// TIA Portal V16 export
// export: Created 2021-11-12T13:31:09.0578565Z, ExportSetting WithDefaults, DisplayName Totally Integrated Automation Portal, DisplayVersion V16 Update 3, DisplayName TIA Portal Version Control Interface, DisplayVersion V16 Update 2, DisplayName TIA Portal Openness, DisplayVersion V16 Update 3, DisplayName SINAMICS Startdrive Advanced, DisplayVersion V16 Update 5, DisplayName SINAMICS Startdrive G130, G150, S120, S150, SINAMICS MV, S210, DisplayVersion V16 Update 5, DisplayName SINAMICS Startdrive G110M, G120, G120C, G120D, G120P, G115D, DisplayVersion V16 Update 5, DisplayName STEP 7 Professional, DisplayVersion V16 Update 3, DisplayName STEP 7 Safety, DisplayVersion V16, DisplayName WinCC UA Professional, DisplayVersion V16 Update 3
FUNCTION_BLOCK "Sfty_Input"   // FB67, F_LAD
{ S7_Optimized_Access := 'TRUE' }
VERSION : 0.1
// Digital and profisafe inputs reading
// stored: AutoNumber true, IsIECCheckEnabled false, UDAEnableTagReadback false
   VAR
      SF_KAS1 { S7_SetPoint := 'True'} : ESTOP1;   // Emergency stop - saw KAS1
      SF_KAS2 { S7_SetPoint := 'True'} : ESTOP1;   // Emergency stop - saw KAS2
      SF_BSN1_2 { S7_SetPoint := 'True'} : ESTOP1;   // Emergency stop - owen BSN1 / BSN2
      SF_SCH1 { S7_SetPoint := 'True'} : ESTOP1;   // Emergency stop - press SCH1
      SF_BSN3 { S7_SetPoint := 'True'} : ESTOP1;   // Emergency stop - owen BSN3
      SF_BSN4_5 { S7_SetPoint := 'True'} : ESTOP1;   // Emergency stop - owen BSN4 / BSN5
      SF_THM1 { S7_SetPoint := 'True'} : ESTOP1;   // Emergency stop - blaster THM1
      SF_THM2 { S7_SetPoint := 'True'} : ESTOP1;   // Emergency stop - blaster THM2
      "SF_1R1-RC01" { S7_SetPoint := 'True'} : ESTOP1;   // Emergency stop - robot 1R1-RC01
      "SF_1R2-RC01" { S7_SetPoint := 'True'} : ESTOP1;   // Emergency stop - robot 1R2-RC01
      "SF_1R3-RC01" { S7_SetPoint := 'True'} : ESTOP1;   // Emergency stop - robot 1R3-RC01
      "SF_1R4-RC01" { S7_SetPoint := 'True'} : ESTOP1;   // Emergency stop - robot 1R4-RC01
      "SF_1R5-RC01" { S7_SetPoint := 'True'} : ESTOP1;   // Emergency stop - robot 1R5-RC01
      "SF_1R6-RC01" { S7_SetPoint := 'True'} : ESTOP1;   // Emergency stop - robot 1R6-RC01
      "SF_2R1-RC01" { S7_SetPoint := 'True'} : ESTOP1;   // Emergency stop - robot 2R1-RC01
      "SF_2R2-RC01" { S7_SetPoint := 'True'} : ESTOP1;   // Emergency stop - robot 2R2-RC01
      "SF_000UH11-SF01_12" { S7_SetPoint := 'True'} : ESTOP1;   // Emergency stop button - panel 000+UH11
      "SF_000UH10-SF01_12" { S7_SetPoint := 'True'} : ESTOP1;   // Emergency stop button - panel 000+UH10
      "SF_100UH11-SF01_12" { S7_SetPoint := 'True'} : ESTOP1;   // Emergency stop button - panel 100+UH11
      "SF_100UH12-SF01_12" { S7_SetPoint := 'True'} : ESTOP1;   // Emergency stop button - panel 100+UH12
      "SF_100UH13-SF01_12" { S7_SetPoint := 'True'} : ESTOP1;   // Emergency stop button - panel 100+UH13
      "SF_100UF01-SF01_12" { S7_SetPoint := 'True'} : ESTOP1;   // Emergency stop button - panel 100+UF01
      "SF_200UH11-SF01_12" { S7_SetPoint := 'True'} : ESTOP1;   // Emergency stop button - panel 200+UH11
      "SF_200UF01-SF01_12" { S7_SetPoint := 'True'} : ESTOP1;   // Emergency stop button - panel 200+UF01
      "SF_210UF01-SF01_12" { S7_SetPoint := 'True'} : ESTOP1;   // Emergency stop button - panel 210+UF01
      "SF_220UF01-SF01_12" { S7_SetPoint := 'True'} : ESTOP1;   // Emergency stop button - panel 220+UF01
      "SF_230UF01-SF01_12" { S7_SetPoint := 'True'} : ESTOP1;   // Emergency stop button - panel 230+UF01
      "SF_300UH11-SF01_12" { S7_SetPoint := 'True'} : ESTOP1;   // Emergency stop button - panel 300+UH11
      "SF_310UH31-SF01_12" { S7_SetPoint := 'True'} : ESTOP1;   // Emergency stop button - panel 300+UH11
      "SF_330UF01-SF01_12" { S7_SetPoint := 'True'} : ESTOP1;   // Emergency stop button - panel 330+UF01
      "SF_400UH11-SF01_12" { S7_SetPoint := 'True'} : ESTOP1;   // Emergency stop button - panel 400+UH11
      "SF_400UH31-SF01_12" { S7_SetPoint := 'True'} : ESTOP1;   // Emergency stop button - panel 400+UH31
      "SF_410UH31-SF01_12" { S7_SetPoint := 'True'} : ESTOP1;   // Emergency stop button - panel 400+UH31
      "SF_420UH31-SF01_12" { S7_SetPoint := 'True'} : ESTOP1;   // Emergency stop button - panel 400+UH31
      "SF_100+RU01-QQ01" { S7_SetPoint := 'True'} : ESTOP1;   // Emergency stop button - gate 100+RU01-QQ01
      "SF_100+RU01-QQ02" { S7_SetPoint := 'True'} : ESTOP1;   // Emergency stop button - gate 100+RU01-QQ02
      "SF_100+RU01-QQ03" { S7_SetPoint := 'True'} : ESTOP1;   // Emergency stop button - gate 100+RU01-QQ03
      "SF_100+RU01-QQ04" { S7_SetPoint := 'True'} : ESTOP1;   // Emergency stop button - gate 100+RU01-QQ04
      "SF_100+RU01-QQ05" { S7_SetPoint := 'True'} : ESTOP1;   // Emergency stop button - gate 100+RU01-QQ05
      "SF_100+RU01-QQ06" { S7_SetPoint := 'True'} : ESTOP1;   // Emergency stop button - gate 100+RU01-QQ06
      "SF_100+RU01-QQ07" { S7_SetPoint := 'True'} : ESTOP1;   // Emergency stop button - gate 100+RU01-QQ07
      "SF_100+RU01-QQ08" { S7_SetPoint := 'True'} : ESTOP1;   // Emergency stop button - gate 100+RU01-QQ08
      "SF_200RU01-QQ01" { S7_SetPoint := 'True'} : ESTOP1;   // Emergency stop button - gate 200RU01-QQ01
      "SF_200RU01-QQ02" { S7_SetPoint := 'True'} : ESTOP1;   // Emergency stop button - gate 200RU01-QQ02
      "SF_200RU01-QQ03" { S7_SetPoint := 'True'} : ESTOP1;   // Emergency stop button - gate 200RU01-QQ03
      "SF_200RU01-QQ04" { S7_SetPoint := 'True'} : ESTOP1;   // Emergency stop button - gate 200RU01-QQ04
      "SF_200RU01-QQ05" { S7_SetPoint := 'True'} : ESTOP1;   // Emergency stop button - gate 200RU01-QQ05
      "SF_100+RU01-QQ01_lock" { S7_SetPoint := 'True'} : ESTOP1;   // Gate is closed and locked - 100+RU01-QQ01
      "SF_100+RU01-QQ02_lock" { S7_SetPoint := 'True'} : ESTOP1;   // Gate is closed and locked - 100+RU01-QQ02
      "SF_100+RU01-QQ03_lock" { S7_SetPoint := 'True'} : ESTOP1;   // Gate is closed and locked - 100+RU01-QQ03
      "SF_100+RU01-QQ04_lock" { S7_SetPoint := 'True'} : ESTOP1;   // Gate is closed and locked - 100+RU01-QQ04
      "SF_100+RU01-QQ05_lock" { S7_SetPoint := 'True'} : ESTOP1;   // Gate is closed and locked - 100+RU01-QQ05
      "SF_100+RU01-QQ06_lock" { S7_SetPoint := 'True'} : ESTOP1;   // Gate is closed and locked - 100+RU01-QQ06
      "SF_100+RU01-QQ07_lock" { S7_SetPoint := 'True'} : ESTOP1;   // Gate is closed and locked - 100+RU01-QQ07
      "SF_100+RU01-QQ08_lock" { S7_SetPoint := 'True'} : ESTOP1;   // Gate is closed and locked - 100+RU01-QQ08
      "SF_200RU01-QQ01_lock" { S7_SetPoint := 'True'} : ESTOP1;   // Gate is closed and locked - 200RU01-QQ01
      "SF_200RU01-QQ02_lock" { S7_SetPoint := 'True'} : ESTOP1;   // Gate is closed and locked - 200RU01-QQ02
      "SF_200RU01-QQ03_lock" { S7_SetPoint := 'True'} : ESTOP1;   // Gate is closed and locked - 200RU01-QQ03
      "SF_200RU01-QQ04_lock" { S7_SetPoint := 'True'} : ESTOP1;   // Gate is closed and locked - 200RU01-QQ04
      "SF_200RU01-QQ05_lock" { S7_SetPoint := 'True'} : ESTOP1;   // Gate is closed and locked - 200RU01-QQ05
      "SF_100+RU01-BG01_close" { S7_SetPoint := 'True'} : ESTOP1;   // Fence closed - 100+RU01-BG01
      "SF_100+RU01-BG02_close" { S7_SetPoint := 'True'} : ESTOP1;   // Fence closed - 100+RU01-BG02
      "SF_200RU01-BG01_close" { S7_SetPoint := 'True'} : ESTOP1;   // Fence closed - 200RU01-BG01
      "SF_100UR01-KG01R" { S7_SetPoint := 'True'} : ESTOP1;   // Light barrier ok - 100UR01-KG01
      "SF_100UR01-KG02R" { S7_SetPoint := 'True'} : ESTOP1;   // Light barrier ok - 100UR01-KG02
   END_VAR
BEGIN

REGION Network 1: *************** Estop suppliers ***************
END_REGION

REGION Network 2: Emergency stop - saw KAS1
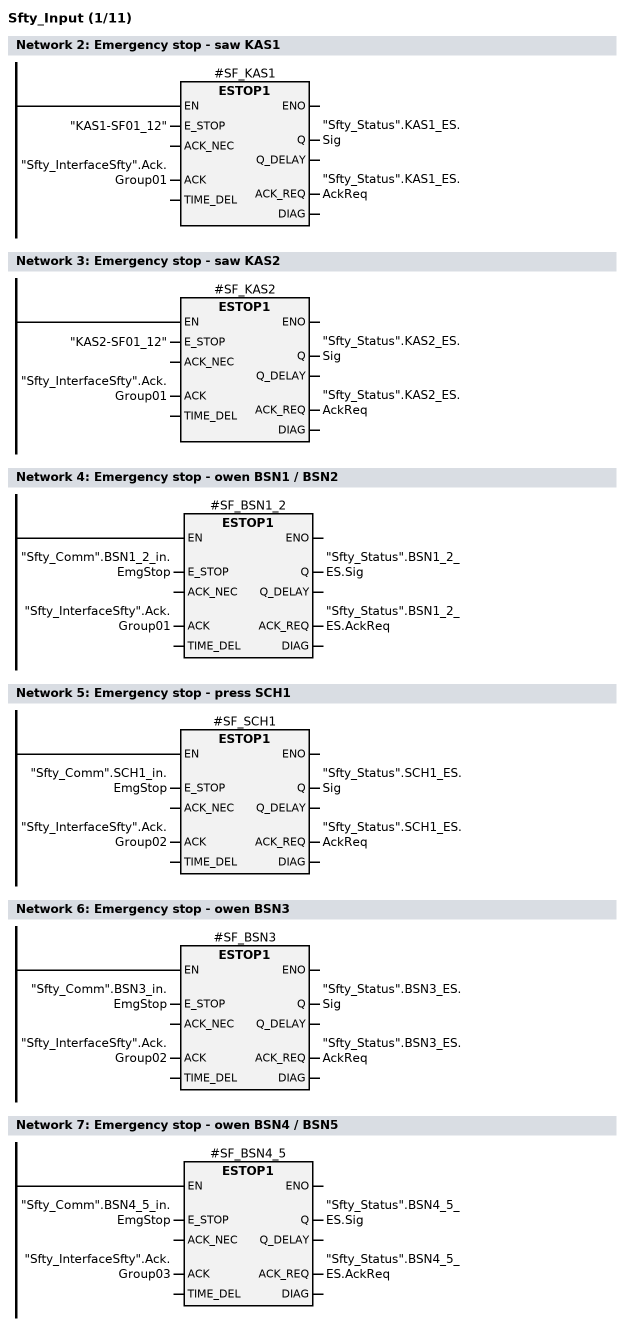
   RUNG wire#powerrail
      #SF_KAS1.ESTOP1(E_STOP := "KAS1-SF01_12", ACK_NEC :=, ACK := "Sfty_InterfaceSfty".Ack.Group01, TIME_DEL :=, Q => "Sfty_Status".KAS1_ES.Sig, Q_DELAY =>, ACK_REQ => "Sfty_Status".KAS1_ES.AckReq, DIAG =>)
   END_RUNG
   // the same network as SCL:
   #SF_KAS1(E_STOP := "KAS1-SF01_12",   // ESTOP1
            ACK := "Sfty_InterfaceSfty".Ack.Group01,
            Q => "Sfty_Status".KAS1_ES.Sig,
            ACK_REQ => "Sfty_Status".KAS1_ES.AckReq);
END_REGION

REGION Network 3: Emergency stop - saw KAS2
   RUNG wire#powerrail
      #SF_KAS2.ESTOP1(E_STOP := "KAS2-SF01_12", ACK_NEC :=, ACK := "Sfty_InterfaceSfty".Ack.Group01, TIME_DEL :=, Q => "Sfty_Status".KAS2_ES.Sig, Q_DELAY =>, ACK_REQ => "Sfty_Status".KAS2_ES.AckReq, DIAG =>)
   END_RUNG
   // the same network as SCL:
   #SF_KAS2(E_STOP := "KAS2-SF01_12",   // ESTOP1
            ACK := "Sfty_InterfaceSfty".Ack.Group01,
            Q => "Sfty_Status".KAS2_ES.Sig,
            ACK_REQ => "Sfty_Status".KAS2_ES.AckReq);
END_REGION

REGION Network 4: Emergency stop - owen BSN1 / BSN2
   RUNG wire#powerrail
      #SF_BSN1_2.ESTOP1(E_STOP := "Sfty_Comm".BSN1_2_in.EmgStop, ACK_NEC :=, ACK := "Sfty_InterfaceSfty".Ack.Group01, TIME_DEL :=, Q => "Sfty_Status".BSN1_2_ES.Sig, Q_DELAY =>, ACK_REQ => "Sfty_Status".BSN1_2_ES.AckReq, DIAG =>)
   END_RUNG
   // the same network as SCL:
   #SF_BSN1_2(E_STOP := "Sfty_Comm".BSN1_2_in.EmgStop,   // ESTOP1
              ACK := "Sfty_InterfaceSfty".Ack.Group01,
              Q => "Sfty_Status".BSN1_2_ES.Sig,
              ACK_REQ => "Sfty_Status".BSN1_2_ES.AckReq);
END_REGION

REGION Network 5: Emergency stop - press SCH1
   RUNG wire#powerrail
      #SF_SCH1.ESTOP1(E_STOP := "Sfty_Comm".SCH1_in.EmgStop, ACK_NEC :=, ACK := "Sfty_InterfaceSfty".Ack.Group02, TIME_DEL :=, Q => "Sfty_Status".SCH1_ES.Sig, Q_DELAY =>, ACK_REQ => "Sfty_Status".SCH1_ES.AckReq, DIAG =>)
   END_RUNG
   // the same network as SCL:
   #SF_SCH1(E_STOP := "Sfty_Comm".SCH1_in.EmgStop,   // ESTOP1
            ACK := "Sfty_InterfaceSfty".Ack.Group02,
            Q => "Sfty_Status".SCH1_ES.Sig,
            ACK_REQ => "Sfty_Status".SCH1_ES.AckReq);
END_REGION

REGION Network 6: Emergency stop - owen BSN3
   RUNG wire#powerrail
      #SF_BSN3.ESTOP1(E_STOP := "Sfty_Comm".BSN3_in.EmgStop, ACK_NEC :=, ACK := "Sfty_InterfaceSfty".Ack.Group02, TIME_DEL :=, Q => "Sfty_Status".BSN3_ES.Sig, Q_DELAY =>, ACK_REQ => "Sfty_Status".BSN3_ES.AckReq, DIAG =>)
   END_RUNG
   // the same network as SCL:
   #SF_BSN3(E_STOP := "Sfty_Comm".BSN3_in.EmgStop,   // ESTOP1
            ACK := "Sfty_InterfaceSfty".Ack.Group02,
            Q => "Sfty_Status".BSN3_ES.Sig,
            ACK_REQ => "Sfty_Status".BSN3_ES.AckReq);
END_REGION

REGION Network 7: Emergency stop - owen BSN4 / BSN5
   RUNG wire#powerrail
      #SF_BSN4_5.ESTOP1(E_STOP := "Sfty_Comm".BSN4_5_in.EmgStop, ACK_NEC :=, ACK := "Sfty_InterfaceSfty".Ack.Group03, TIME_DEL :=, Q => "Sfty_Status".BSN4_5_ES.Sig, Q_DELAY =>, ACK_REQ => "Sfty_Status".BSN4_5_ES.AckReq, DIAG =>)
   END_RUNG
   // the same network as SCL:
   #SF_BSN4_5(E_STOP := "Sfty_Comm".BSN4_5_in.EmgStop,   // ESTOP1
              ACK := "Sfty_InterfaceSfty".Ack.Group03,
              Q => "Sfty_Status".BSN4_5_ES.Sig,
              ACK_REQ => "Sfty_Status".BSN4_5_ES.AckReq);
END_REGION

REGION Network 8: Emergency stop - blaster THM1
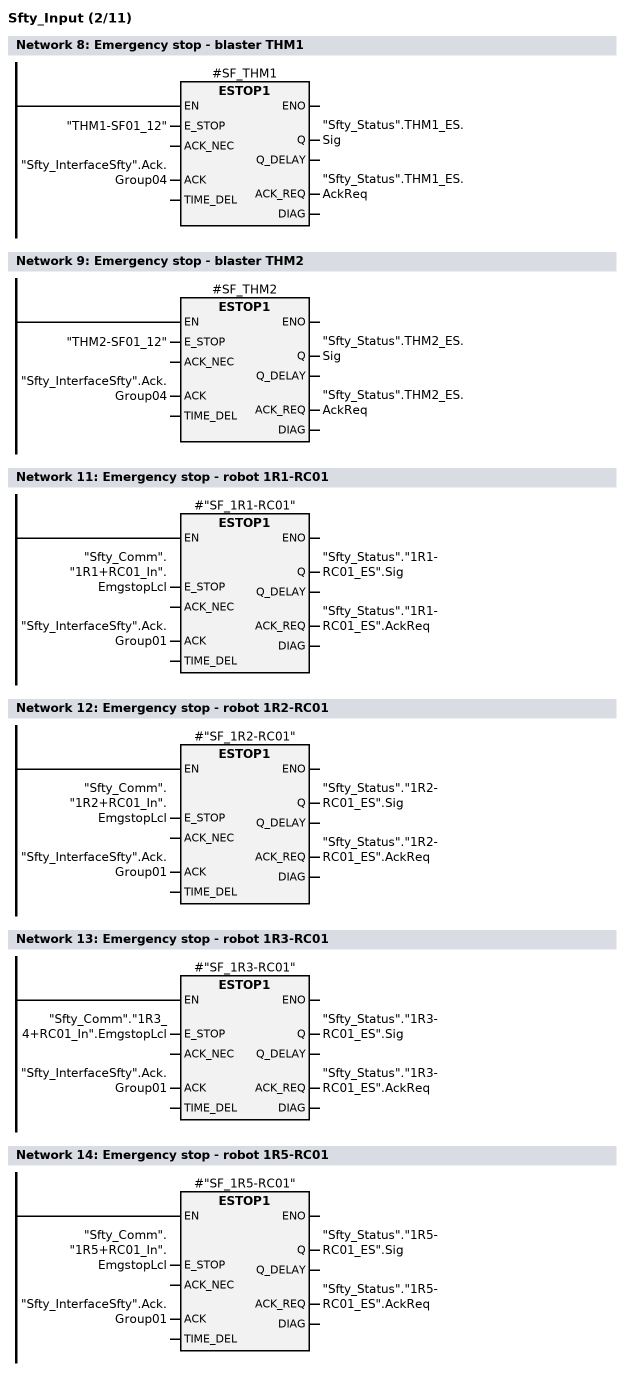
   RUNG wire#powerrail
      #SF_THM1.ESTOP1(E_STOP := "THM1-SF01_12", ACK_NEC :=, ACK := "Sfty_InterfaceSfty".Ack.Group04, TIME_DEL :=, Q => "Sfty_Status".THM1_ES.Sig, Q_DELAY =>, ACK_REQ => "Sfty_Status".THM1_ES.AckReq, DIAG =>)
   END_RUNG
   // the same network as SCL:
   #SF_THM1(E_STOP := "THM1-SF01_12",   // ESTOP1
            ACK := "Sfty_InterfaceSfty".Ack.Group04,
            Q => "Sfty_Status".THM1_ES.Sig,
            ACK_REQ => "Sfty_Status".THM1_ES.AckReq);
END_REGION

REGION Network 9: Emergency stop - blaster THM2
   RUNG wire#powerrail
      #SF_THM2.ESTOP1(E_STOP := "THM2-SF01_12", ACK_NEC :=, ACK := "Sfty_InterfaceSfty".Ack.Group04, TIME_DEL :=, Q => "Sfty_Status".THM2_ES.Sig, Q_DELAY =>, ACK_REQ => "Sfty_Status".THM2_ES.AckReq, DIAG =>)
   END_RUNG
   // the same network as SCL:
   #SF_THM2(E_STOP := "THM2-SF01_12",   // ESTOP1
            ACK := "Sfty_InterfaceSfty".Ack.Group04,
            Q => "Sfty_Status".THM2_ES.Sig,
            ACK_REQ => "Sfty_Status".THM2_ES.AckReq);
END_REGION

REGION Network 10: *************** ESTOP robots ***************
END_REGION

REGION Network 11: Emergency stop - robot 1R1-RC01
   RUNG wire#powerrail
      #"SF_1R1-RC01".ESTOP1(E_STOP := "Sfty_Comm"."1R1+RC01_In".EmgstopLcl, ACK_NEC :=, ACK := "Sfty_InterfaceSfty".Ack.Group01, TIME_DEL :=, Q => "Sfty_Status"."1R1-RC01_ES".Sig, Q_DELAY =>, ACK_REQ => "Sfty_Status"."1R1-RC01_ES".AckReq, DIAG =>)
   END_RUNG
   // the same network as SCL:
   #"SF_1R1-RC01"(E_STOP := "Sfty_Comm"."1R1+RC01_In".EmgstopLcl,   // ESTOP1
                  ACK := "Sfty_InterfaceSfty".Ack.Group01,
                  Q => "Sfty_Status"."1R1-RC01_ES".Sig,
                  ACK_REQ => "Sfty_Status"."1R1-RC01_ES".AckReq);
END_REGION

REGION Network 12: Emergency stop - robot 1R2-RC01
   RUNG wire#powerrail
      #"SF_1R2-RC01".ESTOP1(E_STOP := "Sfty_Comm"."1R2+RC01_In".EmgstopLcl, ACK_NEC :=, ACK := "Sfty_InterfaceSfty".Ack.Group01, TIME_DEL :=, Q => "Sfty_Status"."1R2-RC01_ES".Sig, Q_DELAY =>, ACK_REQ => "Sfty_Status"."1R2-RC01_ES".AckReq, DIAG =>)
   END_RUNG
   // the same network as SCL:
   #"SF_1R2-RC01"(E_STOP := "Sfty_Comm"."1R2+RC01_In".EmgstopLcl,   // ESTOP1
                  ACK := "Sfty_InterfaceSfty".Ack.Group01,
                  Q => "Sfty_Status"."1R2-RC01_ES".Sig,
                  ACK_REQ => "Sfty_Status"."1R2-RC01_ES".AckReq);
END_REGION

REGION Network 13: Emergency stop - robot 1R3-RC01
   RUNG wire#powerrail
      #"SF_1R3-RC01".ESTOP1(E_STOP := "Sfty_Comm"."1R3_4+RC01_In".EmgstopLcl, ACK_NEC :=, ACK := "Sfty_InterfaceSfty".Ack.Group01, TIME_DEL :=, Q => "Sfty_Status"."1R3-RC01_ES".Sig, Q_DELAY =>, ACK_REQ => "Sfty_Status"."1R3-RC01_ES".AckReq, DIAG =>)
   END_RUNG
   // the same network as SCL:
   #"SF_1R3-RC01"(E_STOP := "Sfty_Comm"."1R3_4+RC01_In".EmgstopLcl,   // ESTOP1
                  ACK := "Sfty_InterfaceSfty".Ack.Group01,
                  Q => "Sfty_Status"."1R3-RC01_ES".Sig,
                  ACK_REQ => "Sfty_Status"."1R3-RC01_ES".AckReq);
END_REGION

REGION Network 14: Emergency stop - robot 1R5-RC01
   RUNG wire#powerrail
      #"SF_1R5-RC01".ESTOP1(E_STOP := "Sfty_Comm"."1R5+RC01_In".EmgstopLcl, ACK_NEC :=, ACK := "Sfty_InterfaceSfty".Ack.Group01, TIME_DEL :=, Q => "Sfty_Status"."1R5-RC01_ES".Sig, Q_DELAY =>, ACK_REQ => "Sfty_Status"."1R5-RC01_ES".AckReq, DIAG =>)
   END_RUNG
   // the same network as SCL:
   #"SF_1R5-RC01"(E_STOP := "Sfty_Comm"."1R5+RC01_In".EmgstopLcl,   // ESTOP1
                  ACK := "Sfty_InterfaceSfty".Ack.Group01,
                  Q => "Sfty_Status"."1R5-RC01_ES".Sig,
                  ACK_REQ => "Sfty_Status"."1R5-RC01_ES".AckReq);
END_REGION

REGION Network 15: Emergency stop - robot 1R6-RC01
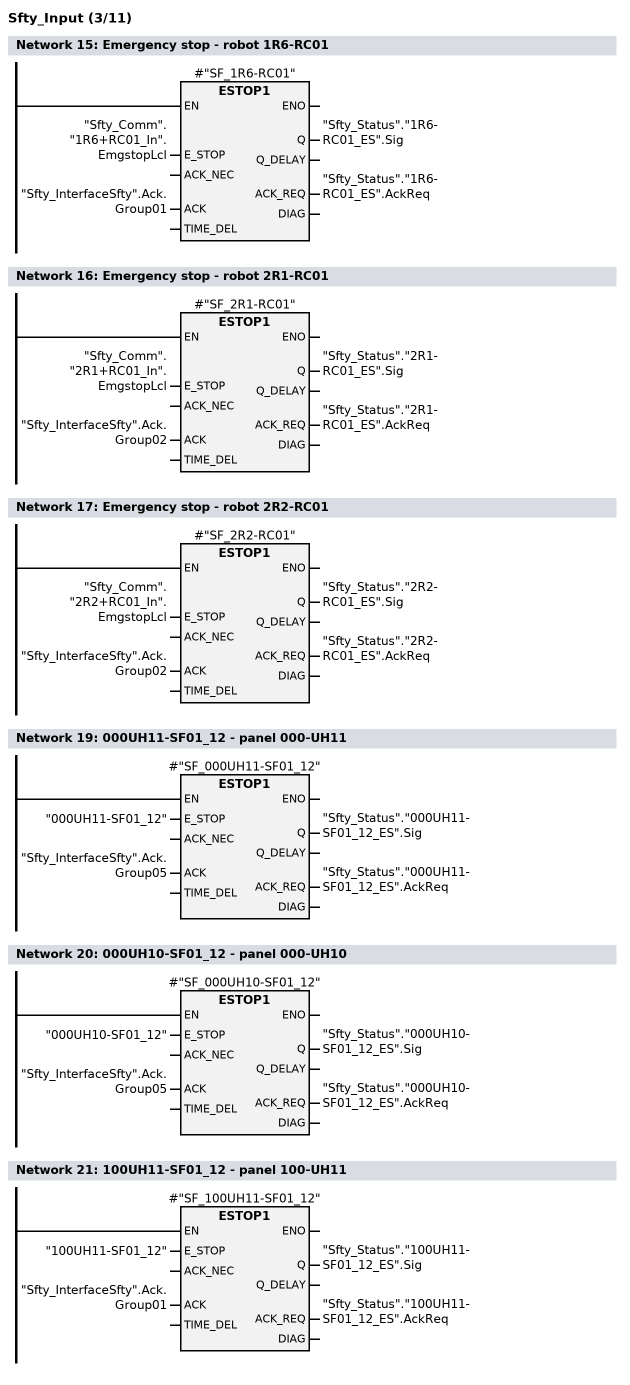
   RUNG wire#powerrail
      #"SF_1R6-RC01".ESTOP1(E_STOP := "Sfty_Comm"."1R6+RC01_In".EmgstopLcl, ACK_NEC :=, ACK := "Sfty_InterfaceSfty".Ack.Group01, TIME_DEL :=, Q => "Sfty_Status"."1R6-RC01_ES".Sig, Q_DELAY =>, ACK_REQ => "Sfty_Status"."1R6-RC01_ES".AckReq, DIAG =>)
   END_RUNG
   // the same network as SCL:
   #"SF_1R6-RC01"(E_STOP := "Sfty_Comm"."1R6+RC01_In".EmgstopLcl,   // ESTOP1
                  ACK := "Sfty_InterfaceSfty".Ack.Group01,
                  Q => "Sfty_Status"."1R6-RC01_ES".Sig,
                  ACK_REQ => "Sfty_Status"."1R6-RC01_ES".AckReq);
END_REGION

REGION Network 16: Emergency stop - robot 2R1-RC01
   RUNG wire#powerrail
      #"SF_2R1-RC01".ESTOP1(E_STOP := "Sfty_Comm"."2R1+RC01_In".EmgstopLcl, ACK_NEC :=, ACK := "Sfty_InterfaceSfty".Ack.Group02, TIME_DEL :=, Q => "Sfty_Status"."2R1-RC01_ES".Sig, Q_DELAY =>, ACK_REQ => "Sfty_Status"."2R1-RC01_ES".AckReq, DIAG =>)
   END_RUNG
   // the same network as SCL:
   #"SF_2R1-RC01"(E_STOP := "Sfty_Comm"."2R1+RC01_In".EmgstopLcl,   // ESTOP1
                  ACK := "Sfty_InterfaceSfty".Ack.Group02,
                  Q => "Sfty_Status"."2R1-RC01_ES".Sig,
                  ACK_REQ => "Sfty_Status"."2R1-RC01_ES".AckReq);
END_REGION

REGION Network 17: Emergency stop - robot 2R2-RC01
   RUNG wire#powerrail
      #"SF_2R2-RC01".ESTOP1(E_STOP := "Sfty_Comm"."2R2+RC01_In".EmgstopLcl, ACK_NEC :=, ACK := "Sfty_InterfaceSfty".Ack.Group02, TIME_DEL :=, Q => "Sfty_Status"."2R2-RC01_ES".Sig, Q_DELAY =>, ACK_REQ => "Sfty_Status"."2R2-RC01_ES".AckReq, DIAG =>)
   END_RUNG
   // the same network as SCL:
   #"SF_2R2-RC01"(E_STOP := "Sfty_Comm"."2R2+RC01_In".EmgstopLcl,   // ESTOP1
                  ACK := "Sfty_InterfaceSfty".Ack.Group02,
                  Q => "Sfty_Status"."2R2-RC01_ES".Sig,
                  ACK_REQ => "Sfty_Status"."2R2-RC01_ES".AckReq);
END_REGION

REGION Network 18: *************** Emergency stop buttons ***************
END_REGION

REGION Network 19: 000UH11-SF01_12 - panel 000-UH11
   RUNG wire#powerrail
      #"SF_000UH11-SF01_12".ESTOP1(E_STOP := "000UH11-SF01_12", ACK_NEC :=, ACK := "Sfty_InterfaceSfty".Ack.Group05, TIME_DEL :=, Q => "Sfty_Status"."000UH11-SF01_12_ES".Sig, Q_DELAY =>, ACK_REQ => "Sfty_Status"."000UH11-SF01_12_ES".AckReq, DIAG =>)
   END_RUNG
   // the same network as SCL:
   #"SF_000UH11-SF01_12"(E_STOP := "000UH11-SF01_12",   // ESTOP1
                         ACK := "Sfty_InterfaceSfty".Ack.Group05,
                         Q => "Sfty_Status"."000UH11-SF01_12_ES".Sig,
                         ACK_REQ => "Sfty_Status"."000UH11-SF01_12_ES".AckReq);
END_REGION

REGION Network 20: 000UH10-SF01_12 - panel 000-UH10
   RUNG wire#powerrail
      #"SF_000UH10-SF01_12".ESTOP1(E_STOP := "000UH10-SF01_12", ACK_NEC :=, ACK := "Sfty_InterfaceSfty".Ack.Group05, TIME_DEL :=, Q => "Sfty_Status"."000UH10-SF01_12_ES".Sig, Q_DELAY =>, ACK_REQ => "Sfty_Status"."000UH10-SF01_12_ES".AckReq, DIAG =>)
   END_RUNG
   // the same network as SCL:
   #"SF_000UH10-SF01_12"(E_STOP := "000UH10-SF01_12",   // ESTOP1
                         ACK := "Sfty_InterfaceSfty".Ack.Group05,
                         Q => "Sfty_Status"."000UH10-SF01_12_ES".Sig,
                         ACK_REQ => "Sfty_Status"."000UH10-SF01_12_ES".AckReq);
END_REGION

REGION Network 21: 100UH11-SF01_12 - panel 100-UH11
   RUNG wire#powerrail
      #"SF_100UH11-SF01_12".ESTOP1(E_STOP := "100UH11-SF01_12", ACK_NEC :=, ACK := "Sfty_InterfaceSfty".Ack.Group01, TIME_DEL :=, Q => "Sfty_Status"."100UH11-SF01_12_ES".Sig, Q_DELAY =>, ACK_REQ => "Sfty_Status"."100UH11-SF01_12_ES".AckReq, DIAG =>)
   END_RUNG
   // the same network as SCL:
   #"SF_100UH11-SF01_12"(E_STOP := "100UH11-SF01_12",   // ESTOP1
                         ACK := "Sfty_InterfaceSfty".Ack.Group01,
                         Q => "Sfty_Status"."100UH11-SF01_12_ES".Sig,
                         ACK_REQ => "Sfty_Status"."100UH11-SF01_12_ES".AckReq);
END_REGION

REGION Network 22: 100UH12-SF01_12 - panel 100-UH12
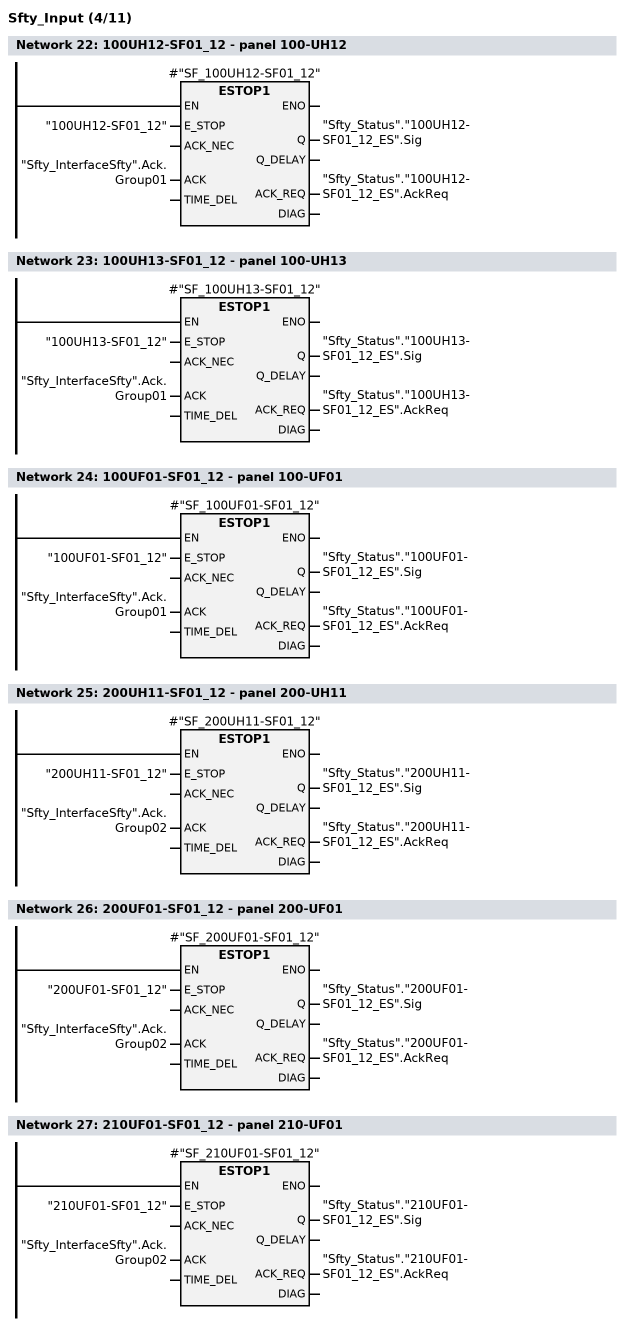
   RUNG wire#powerrail
      #"SF_100UH12-SF01_12".ESTOP1(E_STOP := "100UH12-SF01_12", ACK_NEC :=, ACK := "Sfty_InterfaceSfty".Ack.Group01, TIME_DEL :=, Q => "Sfty_Status"."100UH12-SF01_12_ES".Sig, Q_DELAY =>, ACK_REQ => "Sfty_Status"."100UH12-SF01_12_ES".AckReq, DIAG =>)
   END_RUNG
   // the same network as SCL:
   #"SF_100UH12-SF01_12"(E_STOP := "100UH12-SF01_12",   // ESTOP1
                         ACK := "Sfty_InterfaceSfty".Ack.Group01,
                         Q => "Sfty_Status"."100UH12-SF01_12_ES".Sig,
                         ACK_REQ => "Sfty_Status"."100UH12-SF01_12_ES".AckReq);
END_REGION

REGION Network 23: 100UH13-SF01_12 - panel 100-UH13
   RUNG wire#powerrail
      #"SF_100UH13-SF01_12".ESTOP1(E_STOP := "100UH13-SF01_12", ACK_NEC :=, ACK := "Sfty_InterfaceSfty".Ack.Group01, TIME_DEL :=, Q => "Sfty_Status"."100UH13-SF01_12_ES".Sig, Q_DELAY =>, ACK_REQ => "Sfty_Status"."100UH13-SF01_12_ES".AckReq, DIAG =>)
   END_RUNG
   // the same network as SCL:
   #"SF_100UH13-SF01_12"(E_STOP := "100UH13-SF01_12",   // ESTOP1
                         ACK := "Sfty_InterfaceSfty".Ack.Group01,
                         Q => "Sfty_Status"."100UH13-SF01_12_ES".Sig,
                         ACK_REQ => "Sfty_Status"."100UH13-SF01_12_ES".AckReq);
END_REGION

REGION Network 24: 100UF01-SF01_12 - panel 100-UF01
   RUNG wire#powerrail
      #"SF_100UF01-SF01_12".ESTOP1(E_STOP := "100UF01-SF01_12", ACK_NEC :=, ACK := "Sfty_InterfaceSfty".Ack.Group01, TIME_DEL :=, Q => "Sfty_Status"."100UF01-SF01_12_ES".Sig, Q_DELAY =>, ACK_REQ => "Sfty_Status"."100UF01-SF01_12_ES".AckReq, DIAG =>)
   END_RUNG
   // the same network as SCL:
   #"SF_100UF01-SF01_12"(E_STOP := "100UF01-SF01_12",   // ESTOP1
                         ACK := "Sfty_InterfaceSfty".Ack.Group01,
                         Q => "Sfty_Status"."100UF01-SF01_12_ES".Sig,
                         ACK_REQ => "Sfty_Status"."100UF01-SF01_12_ES".AckReq);
END_REGION

REGION Network 25: 200UH11-SF01_12 - panel 200-UH11
   RUNG wire#powerrail
      #"SF_200UH11-SF01_12".ESTOP1(E_STOP := "200UH11-SF01_12", ACK_NEC :=, ACK := "Sfty_InterfaceSfty".Ack.Group02, TIME_DEL :=, Q => "Sfty_Status"."200UH11-SF01_12_ES".Sig, Q_DELAY =>, ACK_REQ => "Sfty_Status"."200UH11-SF01_12_ES".AckReq, DIAG =>)
   END_RUNG
   // the same network as SCL:
   #"SF_200UH11-SF01_12"(E_STOP := "200UH11-SF01_12",   // ESTOP1
                         ACK := "Sfty_InterfaceSfty".Ack.Group02,
                         Q => "Sfty_Status"."200UH11-SF01_12_ES".Sig,
                         ACK_REQ => "Sfty_Status"."200UH11-SF01_12_ES".AckReq);
END_REGION

REGION Network 26: 200UF01-SF01_12 - panel 200-UF01
   RUNG wire#powerrail
      #"SF_200UF01-SF01_12".ESTOP1(E_STOP := "200UF01-SF01_12", ACK_NEC :=, ACK := "Sfty_InterfaceSfty".Ack.Group02, TIME_DEL :=, Q => "Sfty_Status"."200UF01-SF01_12_ES".Sig, Q_DELAY =>, ACK_REQ => "Sfty_Status"."200UF01-SF01_12_ES".AckReq, DIAG =>)
   END_RUNG
   // the same network as SCL:
   #"SF_200UF01-SF01_12"(E_STOP := "200UF01-SF01_12",   // ESTOP1
                         ACK := "Sfty_InterfaceSfty".Ack.Group02,
                         Q => "Sfty_Status"."200UF01-SF01_12_ES".Sig,
                         ACK_REQ => "Sfty_Status"."200UF01-SF01_12_ES".AckReq);
END_REGION

REGION Network 27: 210UF01-SF01_12 - panel 210-UF01
   RUNG wire#powerrail
      #"SF_210UF01-SF01_12".ESTOP1(E_STOP := "210UF01-SF01_12", ACK_NEC :=, ACK := "Sfty_InterfaceSfty".Ack.Group02, TIME_DEL :=, Q => "Sfty_Status"."210UF01-SF01_12_ES".Sig, Q_DELAY =>, ACK_REQ => "Sfty_Status"."210UF01-SF01_12_ES".AckReq, DIAG =>)
   END_RUNG
   // the same network as SCL:
   #"SF_210UF01-SF01_12"(E_STOP := "210UF01-SF01_12",   // ESTOP1
                         ACK := "Sfty_InterfaceSfty".Ack.Group02,
                         Q => "Sfty_Status"."210UF01-SF01_12_ES".Sig,
                         ACK_REQ => "Sfty_Status"."210UF01-SF01_12_ES".AckReq);
END_REGION

REGION Network 28: 220UF01-SF01_12 - panel 220-UF01
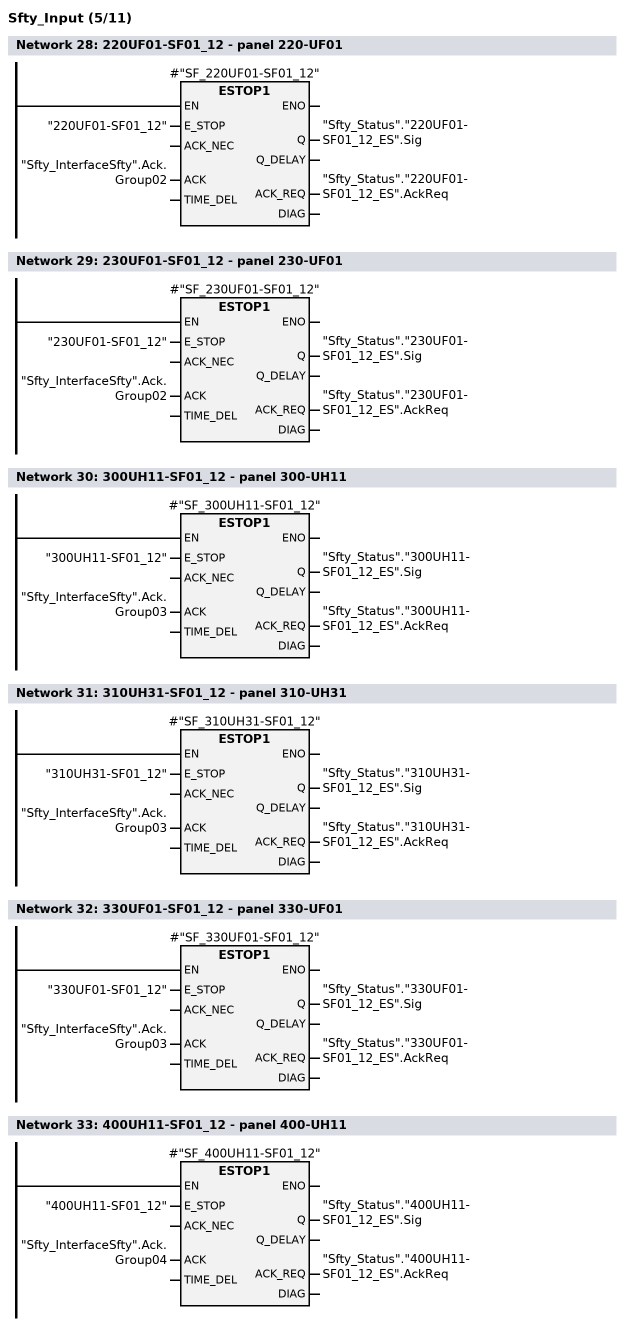
   RUNG wire#powerrail
      #"SF_220UF01-SF01_12".ESTOP1(E_STOP := "220UF01-SF01_12", ACK_NEC :=, ACK := "Sfty_InterfaceSfty".Ack.Group02, TIME_DEL :=, Q => "Sfty_Status"."220UF01-SF01_12_ES".Sig, Q_DELAY =>, ACK_REQ => "Sfty_Status"."220UF01-SF01_12_ES".AckReq, DIAG =>)
   END_RUNG
   // the same network as SCL:
   #"SF_220UF01-SF01_12"(E_STOP := "220UF01-SF01_12",   // ESTOP1
                         ACK := "Sfty_InterfaceSfty".Ack.Group02,
                         Q => "Sfty_Status"."220UF01-SF01_12_ES".Sig,
                         ACK_REQ => "Sfty_Status"."220UF01-SF01_12_ES".AckReq);
END_REGION

REGION Network 29: 230UF01-SF01_12 - panel 230-UF01
   RUNG wire#powerrail
      #"SF_230UF01-SF01_12".ESTOP1(E_STOP := "230UF01-SF01_12", ACK_NEC :=, ACK := "Sfty_InterfaceSfty".Ack.Group02, TIME_DEL :=, Q => "Sfty_Status"."230UF01-SF01_12_ES".Sig, Q_DELAY =>, ACK_REQ => "Sfty_Status"."230UF01-SF01_12_ES".AckReq, DIAG =>)
   END_RUNG
   // the same network as SCL:
   #"SF_230UF01-SF01_12"(E_STOP := "230UF01-SF01_12",   // ESTOP1
                         ACK := "Sfty_InterfaceSfty".Ack.Group02,
                         Q => "Sfty_Status"."230UF01-SF01_12_ES".Sig,
                         ACK_REQ => "Sfty_Status"."230UF01-SF01_12_ES".AckReq);
END_REGION

REGION Network 30: 300UH11-SF01_12 - panel 300-UH11
   RUNG wire#powerrail
      #"SF_300UH11-SF01_12".ESTOP1(E_STOP := "300UH11-SF01_12", ACK_NEC :=, ACK := "Sfty_InterfaceSfty".Ack.Group03, TIME_DEL :=, Q => "Sfty_Status"."300UH11-SF01_12_ES".Sig, Q_DELAY =>, ACK_REQ => "Sfty_Status"."300UH11-SF01_12_ES".AckReq, DIAG =>)
   END_RUNG
   // the same network as SCL:
   #"SF_300UH11-SF01_12"(E_STOP := "300UH11-SF01_12",   // ESTOP1
                         ACK := "Sfty_InterfaceSfty".Ack.Group03,
                         Q => "Sfty_Status"."300UH11-SF01_12_ES".Sig,
                         ACK_REQ => "Sfty_Status"."300UH11-SF01_12_ES".AckReq);
END_REGION

REGION Network 31: 310UH31-SF01_12 - panel 310-UH31
   RUNG wire#powerrail
      #"SF_310UH31-SF01_12".ESTOP1(E_STOP := "310UH31-SF01_12", ACK_NEC :=, ACK := "Sfty_InterfaceSfty".Ack.Group03, TIME_DEL :=, Q => "Sfty_Status"."310UH31-SF01_12_ES".Sig, Q_DELAY =>, ACK_REQ => "Sfty_Status"."310UH31-SF01_12_ES".AckReq, DIAG =>)
   END_RUNG
   // the same network as SCL:
   #"SF_310UH31-SF01_12"(E_STOP := "310UH31-SF01_12",   // ESTOP1
                         ACK := "Sfty_InterfaceSfty".Ack.Group03,
                         Q => "Sfty_Status"."310UH31-SF01_12_ES".Sig,
                         ACK_REQ => "Sfty_Status"."310UH31-SF01_12_ES".AckReq);
END_REGION

REGION Network 32: 330UF01-SF01_12 - panel 330-UF01
   RUNG wire#powerrail
      #"SF_330UF01-SF01_12".ESTOP1(E_STOP := "330UF01-SF01_12", ACK_NEC :=, ACK := "Sfty_InterfaceSfty".Ack.Group03, TIME_DEL :=, Q => "Sfty_Status"."330UF01-SF01_12_ES".Sig, Q_DELAY =>, ACK_REQ => "Sfty_Status"."330UF01-SF01_12_ES".AckReq, DIAG =>)
   END_RUNG
   // the same network as SCL:
   #"SF_330UF01-SF01_12"(E_STOP := "330UF01-SF01_12",   // ESTOP1
                         ACK := "Sfty_InterfaceSfty".Ack.Group03,
                         Q => "Sfty_Status"."330UF01-SF01_12_ES".Sig,
                         ACK_REQ => "Sfty_Status"."330UF01-SF01_12_ES".AckReq);
END_REGION

REGION Network 33: 400UH11-SF01_12 - panel 400-UH11
   RUNG wire#powerrail
      #"SF_400UH11-SF01_12".ESTOP1(E_STOP := "400UH11-SF01_12", ACK_NEC :=, ACK := "Sfty_InterfaceSfty".Ack.Group04, TIME_DEL :=, Q => "Sfty_Status"."400UH11-SF01_12_ES".Sig, Q_DELAY =>, ACK_REQ => "Sfty_Status"."400UH11-SF01_12_ES".AckReq, DIAG =>)
   END_RUNG
   // the same network as SCL:
   #"SF_400UH11-SF01_12"(E_STOP := "400UH11-SF01_12",   // ESTOP1
                         ACK := "Sfty_InterfaceSfty".Ack.Group04,
                         Q => "Sfty_Status"."400UH11-SF01_12_ES".Sig,
                         ACK_REQ => "Sfty_Status"."400UH11-SF01_12_ES".AckReq);
END_REGION

REGION Network 34: 400UH31-SF01_12 - panel 400-UH31
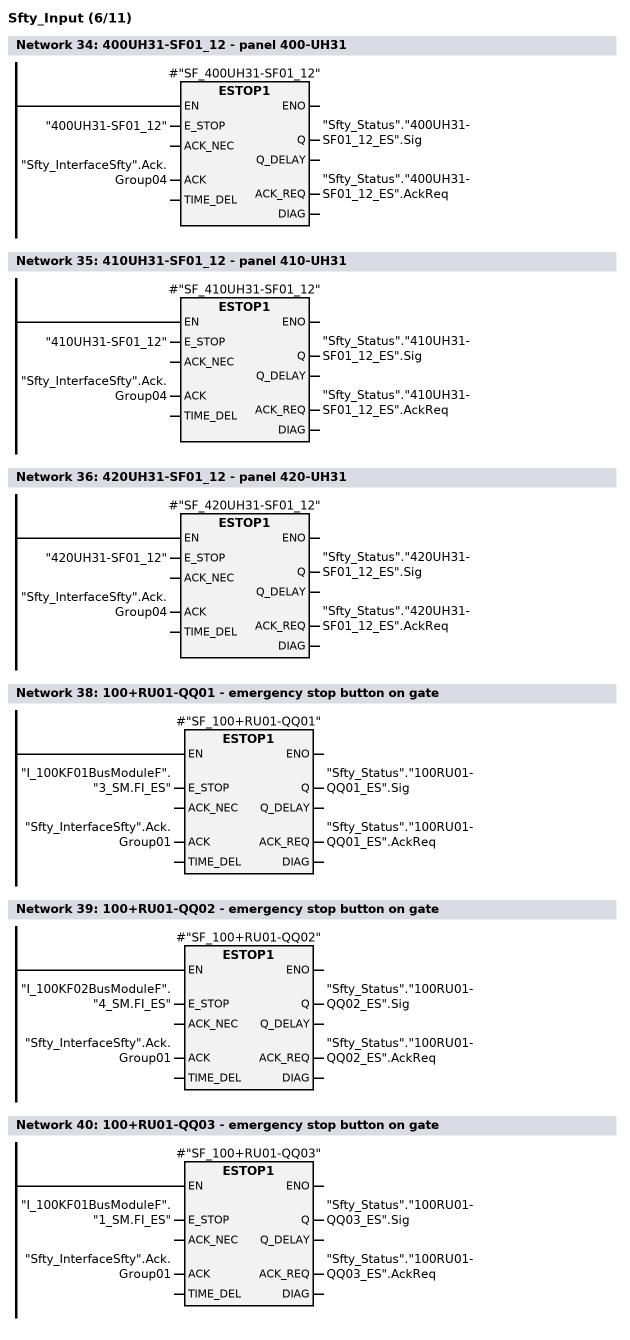
   RUNG wire#powerrail
      #"SF_400UH31-SF01_12".ESTOP1(E_STOP := "400UH31-SF01_12", ACK_NEC :=, ACK := "Sfty_InterfaceSfty".Ack.Group04, TIME_DEL :=, Q => "Sfty_Status"."400UH31-SF01_12_ES".Sig, Q_DELAY =>, ACK_REQ => "Sfty_Status"."400UH31-SF01_12_ES".AckReq, DIAG =>)
   END_RUNG
   // the same network as SCL:
   #"SF_400UH31-SF01_12"(E_STOP := "400UH31-SF01_12",   // ESTOP1
                         ACK := "Sfty_InterfaceSfty".Ack.Group04,
                         Q => "Sfty_Status"."400UH31-SF01_12_ES".Sig,
                         ACK_REQ => "Sfty_Status"."400UH31-SF01_12_ES".AckReq);
END_REGION

REGION Network 35: 410UH31-SF01_12 - panel 410-UH31
   RUNG wire#powerrail
      #"SF_410UH31-SF01_12".ESTOP1(E_STOP := "410UH31-SF01_12", ACK_NEC :=, ACK := "Sfty_InterfaceSfty".Ack.Group04, TIME_DEL :=, Q => "Sfty_Status"."410UH31-SF01_12_ES".Sig, Q_DELAY =>, ACK_REQ => "Sfty_Status"."410UH31-SF01_12_ES".AckReq, DIAG =>)
   END_RUNG
   // the same network as SCL:
   #"SF_410UH31-SF01_12"(E_STOP := "410UH31-SF01_12",   // ESTOP1
                         ACK := "Sfty_InterfaceSfty".Ack.Group04,
                         Q => "Sfty_Status"."410UH31-SF01_12_ES".Sig,
                         ACK_REQ => "Sfty_Status"."410UH31-SF01_12_ES".AckReq);
END_REGION

REGION Network 36: 420UH31-SF01_12 - panel 420-UH31
   RUNG wire#powerrail
      #"SF_420UH31-SF01_12".ESTOP1(E_STOP := "420UH31-SF01_12", ACK_NEC :=, ACK := "Sfty_InterfaceSfty".Ack.Group04, TIME_DEL :=, Q => "Sfty_Status"."420UH31-SF01_12_ES".Sig, Q_DELAY =>, ACK_REQ => "Sfty_Status"."420UH31-SF01_12_ES".AckReq, DIAG =>)
   END_RUNG
   // the same network as SCL:
   #"SF_420UH31-SF01_12"(E_STOP := "420UH31-SF01_12",   // ESTOP1
                         ACK := "Sfty_InterfaceSfty".Ack.Group04,
                         Q => "Sfty_Status"."420UH31-SF01_12_ES".Sig,
                         ACK_REQ => "Sfty_Status"."420UH31-SF01_12_ES".AckReq);
END_REGION

REGION Network 37: *************** Locks emergency stop buttons***************
END_REGION

REGION Network 38: 100+RU01-QQ01 - emergency stop button on gate
   RUNG wire#powerrail
      #"SF_100+RU01-QQ01".ESTOP1(E_STOP := "I_100KF01BusModuleF"."3_SM.FI_ES", ACK_NEC :=, ACK := "Sfty_InterfaceSfty".Ack.Group01, TIME_DEL :=, Q => "Sfty_Status"."100RU01-QQ01_ES".Sig, Q_DELAY =>, ACK_REQ => "Sfty_Status"."100RU01-QQ01_ES".AckReq, DIAG =>)
   END_RUNG
   // the same network as SCL:
   #"SF_100+RU01-QQ01"(E_STOP := "I_100KF01BusModuleF"."3_SM.FI_ES",   // ESTOP1
                       ACK := "Sfty_InterfaceSfty".Ack.Group01,
                       Q => "Sfty_Status"."100RU01-QQ01_ES".Sig,
                       ACK_REQ => "Sfty_Status"."100RU01-QQ01_ES".AckReq);
END_REGION

REGION Network 39: 100+RU01-QQ02 - emergency stop button on gate
   RUNG wire#powerrail
      #"SF_100+RU01-QQ02".ESTOP1(E_STOP := "I_100KF02BusModuleF"."4_SM.FI_ES", ACK_NEC :=, ACK := "Sfty_InterfaceSfty".Ack.Group01, TIME_DEL :=, Q => "Sfty_Status"."100RU01-QQ02_ES".Sig, Q_DELAY =>, ACK_REQ => "Sfty_Status"."100RU01-QQ02_ES".AckReq, DIAG =>)
   END_RUNG
   // the same network as SCL:
   #"SF_100+RU01-QQ02"(E_STOP := "I_100KF02BusModuleF"."4_SM.FI_ES",   // ESTOP1
                       ACK := "Sfty_InterfaceSfty".Ack.Group01,
                       Q => "Sfty_Status"."100RU01-QQ02_ES".Sig,
                       ACK_REQ => "Sfty_Status"."100RU01-QQ02_ES".AckReq);
END_REGION

REGION Network 40: 100+RU01-QQ03 - emergency stop button on gate
   RUNG wire#powerrail
      #"SF_100+RU01-QQ03".ESTOP1(E_STOP := "I_100KF01BusModuleF"."1_SM.FI_ES", ACK_NEC :=, ACK := "Sfty_InterfaceSfty".Ack.Group01, TIME_DEL :=, Q => "Sfty_Status"."100RU01-QQ03_ES".Sig, Q_DELAY =>, ACK_REQ => "Sfty_Status"."100RU01-QQ03_ES".AckReq, DIAG =>)
   END_RUNG
   // the same network as SCL:
   #"SF_100+RU01-QQ03"(E_STOP := "I_100KF01BusModuleF"."1_SM.FI_ES",   // ESTOP1
                       ACK := "Sfty_InterfaceSfty".Ack.Group01,
                       Q => "Sfty_Status"."100RU01-QQ03_ES".Sig,
                       ACK_REQ => "Sfty_Status"."100RU01-QQ03_ES".AckReq);
END_REGION

REGION Network 41: 100+RU01-QQ04 - emergency stop button on gate
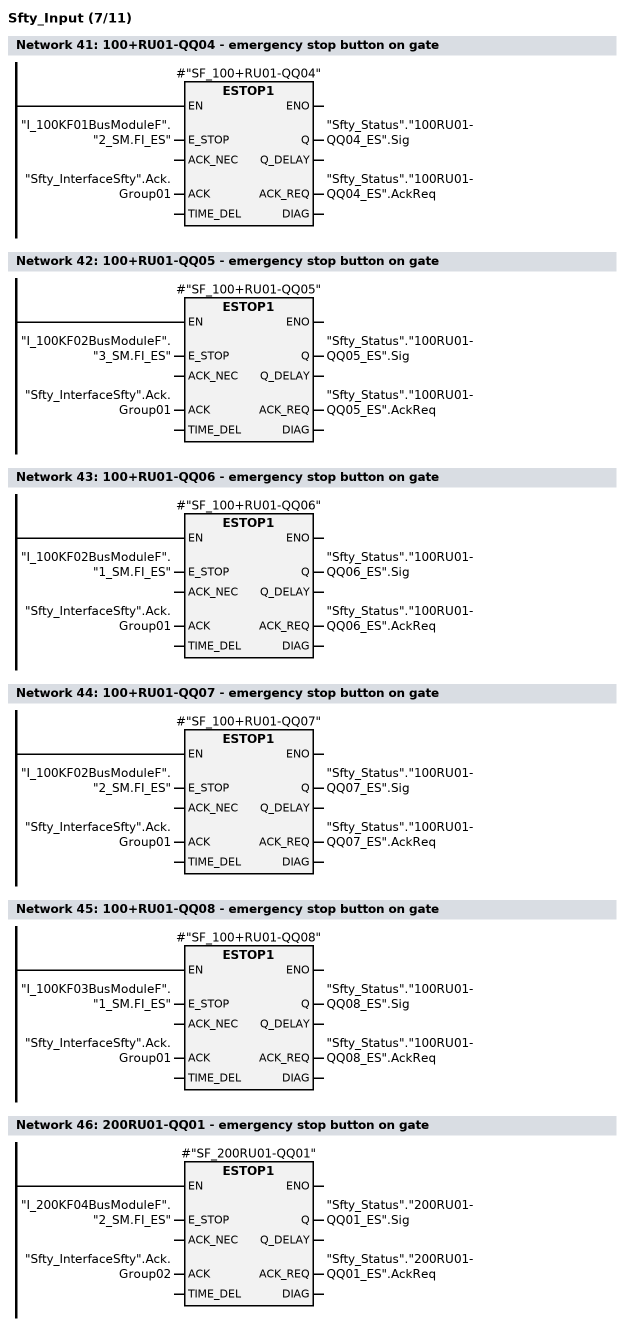
   RUNG wire#powerrail
      #"SF_100+RU01-QQ04".ESTOP1(E_STOP := "I_100KF01BusModuleF"."2_SM.FI_ES", ACK_NEC :=, ACK := "Sfty_InterfaceSfty".Ack.Group01, TIME_DEL :=, Q => "Sfty_Status"."100RU01-QQ04_ES".Sig, Q_DELAY =>, ACK_REQ => "Sfty_Status"."100RU01-QQ04_ES".AckReq, DIAG =>)
   END_RUNG
   // the same network as SCL:
   #"SF_100+RU01-QQ04"(E_STOP := "I_100KF01BusModuleF"."2_SM.FI_ES",   // ESTOP1
                       ACK := "Sfty_InterfaceSfty".Ack.Group01,
                       Q => "Sfty_Status"."100RU01-QQ04_ES".Sig,
                       ACK_REQ => "Sfty_Status"."100RU01-QQ04_ES".AckReq);
END_REGION

REGION Network 42: 100+RU01-QQ05 - emergency stop button on gate
   RUNG wire#powerrail
      #"SF_100+RU01-QQ05".ESTOP1(E_STOP := "I_100KF02BusModuleF"."3_SM.FI_ES", ACK_NEC :=, ACK := "Sfty_InterfaceSfty".Ack.Group01, TIME_DEL :=, Q => "Sfty_Status"."100RU01-QQ05_ES".Sig, Q_DELAY =>, ACK_REQ => "Sfty_Status"."100RU01-QQ05_ES".AckReq, DIAG =>)
   END_RUNG
   // the same network as SCL:
   #"SF_100+RU01-QQ05"(E_STOP := "I_100KF02BusModuleF"."3_SM.FI_ES",   // ESTOP1
                       ACK := "Sfty_InterfaceSfty".Ack.Group01,
                       Q => "Sfty_Status"."100RU01-QQ05_ES".Sig,
                       ACK_REQ => "Sfty_Status"."100RU01-QQ05_ES".AckReq);
END_REGION

REGION Network 43: 100+RU01-QQ06 - emergency stop button on gate
   RUNG wire#powerrail
      #"SF_100+RU01-QQ06".ESTOP1(E_STOP := "I_100KF02BusModuleF"."1_SM.FI_ES", ACK_NEC :=, ACK := "Sfty_InterfaceSfty".Ack.Group01, TIME_DEL :=, Q => "Sfty_Status"."100RU01-QQ06_ES".Sig, Q_DELAY =>, ACK_REQ => "Sfty_Status"."100RU01-QQ06_ES".AckReq, DIAG =>)
   END_RUNG
   // the same network as SCL:
   #"SF_100+RU01-QQ06"(E_STOP := "I_100KF02BusModuleF"."1_SM.FI_ES",   // ESTOP1
                       ACK := "Sfty_InterfaceSfty".Ack.Group01,
                       Q => "Sfty_Status"."100RU01-QQ06_ES".Sig,
                       ACK_REQ => "Sfty_Status"."100RU01-QQ06_ES".AckReq);
END_REGION

REGION Network 44: 100+RU01-QQ07 - emergency stop button on gate
   RUNG wire#powerrail
      #"SF_100+RU01-QQ07".ESTOP1(E_STOP := "I_100KF02BusModuleF"."2_SM.FI_ES", ACK_NEC :=, ACK := "Sfty_InterfaceSfty".Ack.Group01, TIME_DEL :=, Q => "Sfty_Status"."100RU01-QQ07_ES".Sig, Q_DELAY =>, ACK_REQ => "Sfty_Status"."100RU01-QQ07_ES".AckReq, DIAG =>)
   END_RUNG
   // the same network as SCL:
   #"SF_100+RU01-QQ07"(E_STOP := "I_100KF02BusModuleF"."2_SM.FI_ES",   // ESTOP1
                       ACK := "Sfty_InterfaceSfty".Ack.Group01,
                       Q => "Sfty_Status"."100RU01-QQ07_ES".Sig,
                       ACK_REQ => "Sfty_Status"."100RU01-QQ07_ES".AckReq);
END_REGION

REGION Network 45: 100+RU01-QQ08 - emergency stop button on gate
   RUNG wire#powerrail
      #"SF_100+RU01-QQ08".ESTOP1(E_STOP := "I_100KF03BusModuleF"."1_SM.FI_ES", ACK_NEC :=, ACK := "Sfty_InterfaceSfty".Ack.Group01, TIME_DEL :=, Q => "Sfty_Status"."100RU01-QQ08_ES".Sig, Q_DELAY =>, ACK_REQ => "Sfty_Status"."100RU01-QQ08_ES".AckReq, DIAG =>)
   END_RUNG
   // the same network as SCL:
   #"SF_100+RU01-QQ08"(E_STOP := "I_100KF03BusModuleF"."1_SM.FI_ES",   // ESTOP1
                       ACK := "Sfty_InterfaceSfty".Ack.Group01,
                       Q => "Sfty_Status"."100RU01-QQ08_ES".Sig,
                       ACK_REQ => "Sfty_Status"."100RU01-QQ08_ES".AckReq);
END_REGION

REGION Network 46: 200RU01-QQ01 - emergency stop button on gate
   RUNG wire#powerrail
      #"SF_200RU01-QQ01".ESTOP1(E_STOP := "I_200KF04BusModuleF"."2_SM.FI_ES", ACK_NEC :=, ACK := "Sfty_InterfaceSfty".Ack.Group02, TIME_DEL :=, Q => "Sfty_Status"."200RU01-QQ01_ES".Sig, Q_DELAY =>, ACK_REQ => "Sfty_Status"."200RU01-QQ01_ES".AckReq, DIAG =>)
   END_RUNG
   // the same network as SCL:
   #"SF_200RU01-QQ01"(E_STOP := "I_200KF04BusModuleF"."2_SM.FI_ES",   // ESTOP1
                      ACK := "Sfty_InterfaceSfty".Ack.Group02,
                      Q => "Sfty_Status"."200RU01-QQ01_ES".Sig,
                      ACK_REQ => "Sfty_Status"."200RU01-QQ01_ES".AckReq);
END_REGION

REGION Network 47: 200RU01-QQ02 - emergency stop button on gate
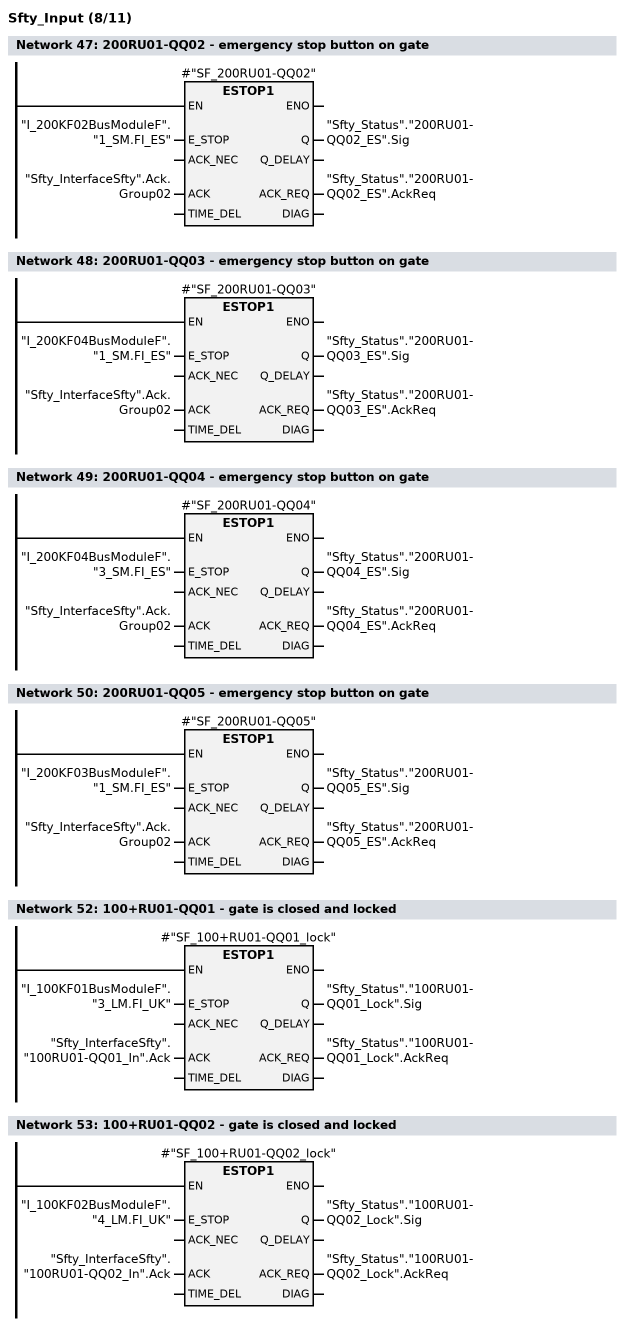
   RUNG wire#powerrail
      #"SF_200RU01-QQ02".ESTOP1(E_STOP := "I_200KF02BusModuleF"."1_SM.FI_ES", ACK_NEC :=, ACK := "Sfty_InterfaceSfty".Ack.Group02, TIME_DEL :=, Q => "Sfty_Status"."200RU01-QQ02_ES".Sig, Q_DELAY =>, ACK_REQ => "Sfty_Status"."200RU01-QQ02_ES".AckReq, DIAG =>)
   END_RUNG
   // the same network as SCL:
   #"SF_200RU01-QQ02"(E_STOP := "I_200KF02BusModuleF"."1_SM.FI_ES",   // ESTOP1
                      ACK := "Sfty_InterfaceSfty".Ack.Group02,
                      Q => "Sfty_Status"."200RU01-QQ02_ES".Sig,
                      ACK_REQ => "Sfty_Status"."200RU01-QQ02_ES".AckReq);
END_REGION

REGION Network 48: 200RU01-QQ03 - emergency stop button on gate
   RUNG wire#powerrail
      #"SF_200RU01-QQ03".ESTOP1(E_STOP := "I_200KF04BusModuleF"."1_SM.FI_ES", ACK_NEC :=, ACK := "Sfty_InterfaceSfty".Ack.Group02, TIME_DEL :=, Q => "Sfty_Status"."200RU01-QQ03_ES".Sig, Q_DELAY =>, ACK_REQ => "Sfty_Status"."200RU01-QQ03_ES".AckReq, DIAG =>)
   END_RUNG
   // the same network as SCL:
   #"SF_200RU01-QQ03"(E_STOP := "I_200KF04BusModuleF"."1_SM.FI_ES",   // ESTOP1
                      ACK := "Sfty_InterfaceSfty".Ack.Group02,
                      Q => "Sfty_Status"."200RU01-QQ03_ES".Sig,
                      ACK_REQ => "Sfty_Status"."200RU01-QQ03_ES".AckReq);
END_REGION

REGION Network 49: 200RU01-QQ04 - emergency stop button on gate
   RUNG wire#powerrail
      #"SF_200RU01-QQ04".ESTOP1(E_STOP := "I_200KF04BusModuleF"."3_SM.FI_ES", ACK_NEC :=, ACK := "Sfty_InterfaceSfty".Ack.Group02, TIME_DEL :=, Q => "Sfty_Status"."200RU01-QQ04_ES".Sig, Q_DELAY =>, ACK_REQ => "Sfty_Status"."200RU01-QQ04_ES".AckReq, DIAG =>)
   END_RUNG
   // the same network as SCL:
   #"SF_200RU01-QQ04"(E_STOP := "I_200KF04BusModuleF"."3_SM.FI_ES",   // ESTOP1
                      ACK := "Sfty_InterfaceSfty".Ack.Group02,
                      Q => "Sfty_Status"."200RU01-QQ04_ES".Sig,
                      ACK_REQ => "Sfty_Status"."200RU01-QQ04_ES".AckReq);
END_REGION

REGION Network 50: 200RU01-QQ05 - emergency stop button on gate
   RUNG wire#powerrail
      #"SF_200RU01-QQ05".ESTOP1(E_STOP := "I_200KF03BusModuleF"."1_SM.FI_ES", ACK_NEC :=, ACK := "Sfty_InterfaceSfty".Ack.Group02, TIME_DEL :=, Q => "Sfty_Status"."200RU01-QQ05_ES".Sig, Q_DELAY =>, ACK_REQ => "Sfty_Status"."200RU01-QQ05_ES".AckReq, DIAG =>)
   END_RUNG
   // the same network as SCL:
   #"SF_200RU01-QQ05"(E_STOP := "I_200KF03BusModuleF"."1_SM.FI_ES",   // ESTOP1
                      ACK := "Sfty_InterfaceSfty".Ack.Group02,
                      Q => "Sfty_Status"."200RU01-QQ05_ES".Sig,
                      ACK_REQ => "Sfty_Status"."200RU01-QQ05_ES".AckReq);
END_REGION

REGION Network 51: *************** Gates are Locks***************
END_REGION

REGION Network 52: 100+RU01-QQ01 - gate is closed and locked
   RUNG wire#powerrail
      #"SF_100+RU01-QQ01_lock".ESTOP1(E_STOP := "I_100KF01BusModuleF"."3_LM.FI_UK", ACK_NEC :=, ACK := "Sfty_InterfaceSfty"."100RU01-QQ01_In".Ack, TIME_DEL :=, Q => "Sfty_Status"."100RU01-QQ01_Lock".Sig, Q_DELAY =>, ACK_REQ => "Sfty_Status"."100RU01-QQ01_Lock".AckReq, DIAG =>)
   END_RUNG
   // the same network as SCL:
   #"SF_100+RU01-QQ01_lock"(E_STOP := "I_100KF01BusModuleF"."3_LM.FI_UK",   // ESTOP1
                           ACK := "Sfty_InterfaceSfty"."100RU01-QQ01_In".Ack,
                           Q => "Sfty_Status"."100RU01-QQ01_Lock".Sig,
                           ACK_REQ => "Sfty_Status"."100RU01-QQ01_Lock".AckReq);
END_REGION

REGION Network 53: 100+RU01-QQ02 - gate is closed and locked
   RUNG wire#powerrail
      #"SF_100+RU01-QQ02_lock".ESTOP1(E_STOP := "I_100KF02BusModuleF"."4_LM.FI_UK", ACK_NEC :=, ACK := "Sfty_InterfaceSfty"."100RU01-QQ02_In".Ack, TIME_DEL :=, Q => "Sfty_Status"."100RU01-QQ02_Lock".Sig, Q_DELAY =>, ACK_REQ => "Sfty_Status"."100RU01-QQ02_Lock".AckReq, DIAG =>)
   END_RUNG
   // the same network as SCL:
   #"SF_100+RU01-QQ02_lock"(E_STOP := "I_100KF02BusModuleF"."4_LM.FI_UK",   // ESTOP1
                           ACK := "Sfty_InterfaceSfty"."100RU01-QQ02_In".Ack,
                           Q => "Sfty_Status"."100RU01-QQ02_Lock".Sig,
                           ACK_REQ => "Sfty_Status"."100RU01-QQ02_Lock".AckReq);
END_REGION

REGION Network 54: 100+RU01-QQ03 - gate is closed and locked
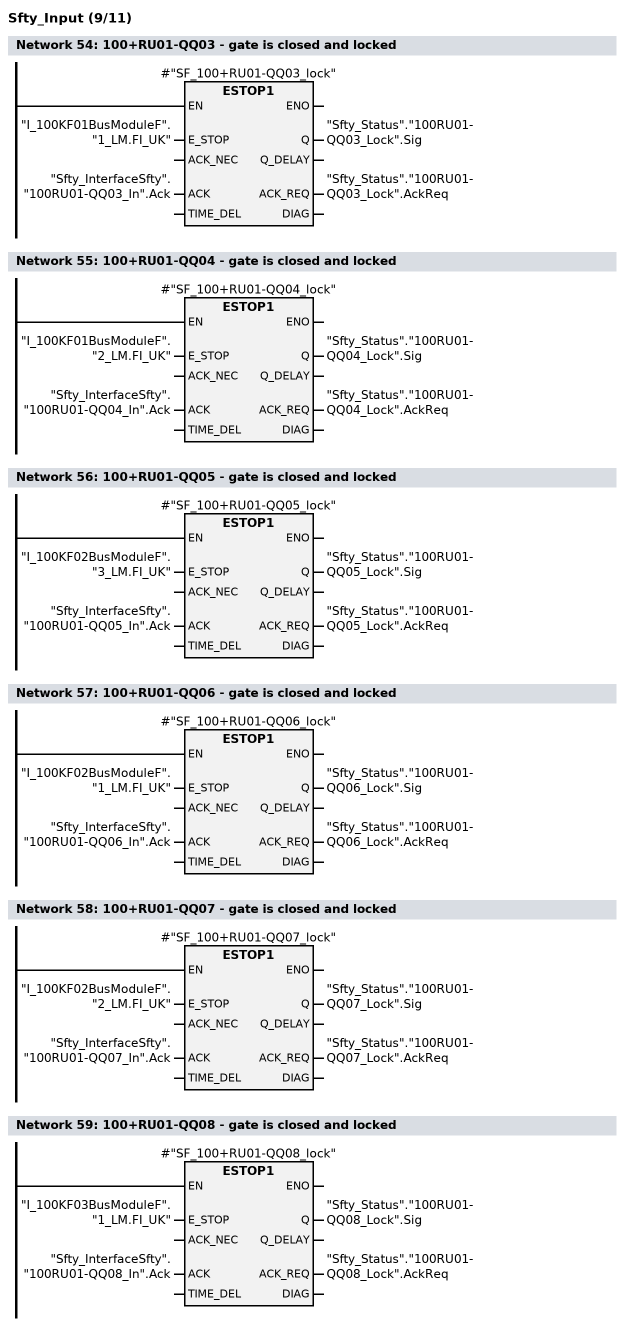
   RUNG wire#powerrail
      #"SF_100+RU01-QQ03_lock".ESTOP1(E_STOP := "I_100KF01BusModuleF"."1_LM.FI_UK", ACK_NEC :=, ACK := "Sfty_InterfaceSfty"."100RU01-QQ03_In".Ack, TIME_DEL :=, Q => "Sfty_Status"."100RU01-QQ03_Lock".Sig, Q_DELAY =>, ACK_REQ => "Sfty_Status"."100RU01-QQ03_Lock".AckReq, DIAG =>)
   END_RUNG
   // the same network as SCL:
   #"SF_100+RU01-QQ03_lock"(E_STOP := "I_100KF01BusModuleF"."1_LM.FI_UK",   // ESTOP1
                           ACK := "Sfty_InterfaceSfty"."100RU01-QQ03_In".Ack,
                           Q => "Sfty_Status"."100RU01-QQ03_Lock".Sig,
                           ACK_REQ => "Sfty_Status"."100RU01-QQ03_Lock".AckReq);
END_REGION

REGION Network 55: 100+RU01-QQ04 - gate is closed and locked
   RUNG wire#powerrail
      #"SF_100+RU01-QQ04_lock".ESTOP1(E_STOP := "I_100KF01BusModuleF"."2_LM.FI_UK", ACK_NEC :=, ACK := "Sfty_InterfaceSfty"."100RU01-QQ04_In".Ack, TIME_DEL :=, Q => "Sfty_Status"."100RU01-QQ04_Lock".Sig, Q_DELAY =>, ACK_REQ => "Sfty_Status"."100RU01-QQ04_Lock".AckReq, DIAG =>)
   END_RUNG
   // the same network as SCL:
   #"SF_100+RU01-QQ04_lock"(E_STOP := "I_100KF01BusModuleF"."2_LM.FI_UK",   // ESTOP1
                           ACK := "Sfty_InterfaceSfty"."100RU01-QQ04_In".Ack,
                           Q => "Sfty_Status"."100RU01-QQ04_Lock".Sig,
                           ACK_REQ => "Sfty_Status"."100RU01-QQ04_Lock".AckReq);
END_REGION

REGION Network 56: 100+RU01-QQ05 - gate is closed and locked
   RUNG wire#powerrail
      #"SF_100+RU01-QQ05_lock".ESTOP1(E_STOP := "I_100KF02BusModuleF"."3_LM.FI_UK", ACK_NEC :=, ACK := "Sfty_InterfaceSfty"."100RU01-QQ05_In".Ack, TIME_DEL :=, Q => "Sfty_Status"."100RU01-QQ05_Lock".Sig, Q_DELAY =>, ACK_REQ => "Sfty_Status"."100RU01-QQ05_Lock".AckReq, DIAG =>)
   END_RUNG
   // the same network as SCL:
   #"SF_100+RU01-QQ05_lock"(E_STOP := "I_100KF02BusModuleF"."3_LM.FI_UK",   // ESTOP1
                           ACK := "Sfty_InterfaceSfty"."100RU01-QQ05_In".Ack,
                           Q => "Sfty_Status"."100RU01-QQ05_Lock".Sig,
                           ACK_REQ => "Sfty_Status"."100RU01-QQ05_Lock".AckReq);
END_REGION

REGION Network 57: 100+RU01-QQ06 - gate is closed and locked
   RUNG wire#powerrail
      #"SF_100+RU01-QQ06_lock".ESTOP1(E_STOP := "I_100KF02BusModuleF"."1_LM.FI_UK", ACK_NEC :=, ACK := "Sfty_InterfaceSfty"."100RU01-QQ06_In".Ack, TIME_DEL :=, Q => "Sfty_Status"."100RU01-QQ06_Lock".Sig, Q_DELAY =>, ACK_REQ => "Sfty_Status"."100RU01-QQ06_Lock".AckReq, DIAG =>)
   END_RUNG
   // the same network as SCL:
   #"SF_100+RU01-QQ06_lock"(E_STOP := "I_100KF02BusModuleF"."1_LM.FI_UK",   // ESTOP1
                           ACK := "Sfty_InterfaceSfty"."100RU01-QQ06_In".Ack,
                           Q => "Sfty_Status"."100RU01-QQ06_Lock".Sig,
                           ACK_REQ => "Sfty_Status"."100RU01-QQ06_Lock".AckReq);
END_REGION

REGION Network 58: 100+RU01-QQ07 - gate is closed and locked
   RUNG wire#powerrail
      #"SF_100+RU01-QQ07_lock".ESTOP1(E_STOP := "I_100KF02BusModuleF"."2_LM.FI_UK", ACK_NEC :=, ACK := "Sfty_InterfaceSfty"."100RU01-QQ07_In".Ack, TIME_DEL :=, Q => "Sfty_Status"."100RU01-QQ07_Lock".Sig, Q_DELAY =>, ACK_REQ => "Sfty_Status"."100RU01-QQ07_Lock".AckReq, DIAG =>)
   END_RUNG
   // the same network as SCL:
   #"SF_100+RU01-QQ07_lock"(E_STOP := "I_100KF02BusModuleF"."2_LM.FI_UK",   // ESTOP1
                           ACK := "Sfty_InterfaceSfty"."100RU01-QQ07_In".Ack,
                           Q => "Sfty_Status"."100RU01-QQ07_Lock".Sig,
                           ACK_REQ => "Sfty_Status"."100RU01-QQ07_Lock".AckReq);
END_REGION

REGION Network 59: 100+RU01-QQ08 - gate is closed and locked
   RUNG wire#powerrail
      #"SF_100+RU01-QQ08_lock".ESTOP1(E_STOP := "I_100KF03BusModuleF"."1_LM.FI_UK", ACK_NEC :=, ACK := "Sfty_InterfaceSfty"."100RU01-QQ08_In".Ack, TIME_DEL :=, Q => "Sfty_Status"."100RU01-QQ08_Lock".Sig, Q_DELAY =>, ACK_REQ => "Sfty_Status"."100RU01-QQ08_Lock".AckReq, DIAG =>)
   END_RUNG
   // the same network as SCL:
   #"SF_100+RU01-QQ08_lock"(E_STOP := "I_100KF03BusModuleF"."1_LM.FI_UK",   // ESTOP1
                           ACK := "Sfty_InterfaceSfty"."100RU01-QQ08_In".Ack,
                           Q => "Sfty_Status"."100RU01-QQ08_Lock".Sig,
                           ACK_REQ => "Sfty_Status"."100RU01-QQ08_Lock".AckReq);
END_REGION

REGION Network 60: 200RU01-QQ01 - gate is closed and locked
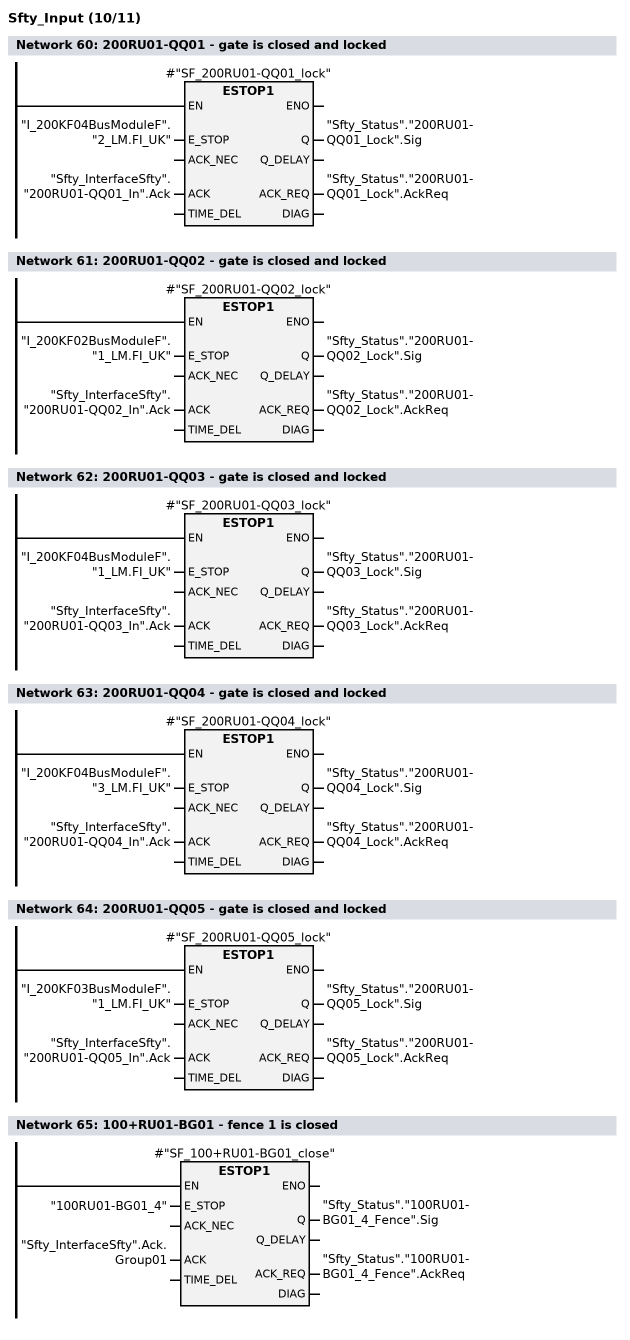
   RUNG wire#powerrail
      #"SF_200RU01-QQ01_lock".ESTOP1(E_STOP := "I_200KF04BusModuleF"."2_LM.FI_UK", ACK_NEC :=, ACK := "Sfty_InterfaceSfty"."200RU01-QQ01_In".Ack, TIME_DEL :=, Q => "Sfty_Status"."200RU01-QQ01_Lock".Sig, Q_DELAY =>, ACK_REQ => "Sfty_Status"."200RU01-QQ01_Lock".AckReq, DIAG =>)
   END_RUNG
   // the same network as SCL:
   #"SF_200RU01-QQ01_lock"(E_STOP := "I_200KF04BusModuleF"."2_LM.FI_UK",   // ESTOP1
                           ACK := "Sfty_InterfaceSfty"."200RU01-QQ01_In".Ack,
                           Q => "Sfty_Status"."200RU01-QQ01_Lock".Sig,
                           ACK_REQ => "Sfty_Status"."200RU01-QQ01_Lock".AckReq);
END_REGION

REGION Network 61: 200RU01-QQ02 - gate is closed and locked
   RUNG wire#powerrail
      #"SF_200RU01-QQ02_lock".ESTOP1(E_STOP := "I_200KF02BusModuleF"."1_LM.FI_UK", ACK_NEC :=, ACK := "Sfty_InterfaceSfty"."200RU01-QQ02_In".Ack, TIME_DEL :=, Q => "Sfty_Status"."200RU01-QQ02_Lock".Sig, Q_DELAY =>, ACK_REQ => "Sfty_Status"."200RU01-QQ02_Lock".AckReq, DIAG =>)
   END_RUNG
   // the same network as SCL:
   #"SF_200RU01-QQ02_lock"(E_STOP := "I_200KF02BusModuleF"."1_LM.FI_UK",   // ESTOP1
                           ACK := "Sfty_InterfaceSfty"."200RU01-QQ02_In".Ack,
                           Q => "Sfty_Status"."200RU01-QQ02_Lock".Sig,
                           ACK_REQ => "Sfty_Status"."200RU01-QQ02_Lock".AckReq);
END_REGION

REGION Network 62: 200RU01-QQ03 - gate is closed and locked
   RUNG wire#powerrail
      #"SF_200RU01-QQ03_lock".ESTOP1(E_STOP := "I_200KF04BusModuleF"."1_LM.FI_UK", ACK_NEC :=, ACK := "Sfty_InterfaceSfty"."200RU01-QQ03_In".Ack, TIME_DEL :=, Q => "Sfty_Status"."200RU01-QQ03_Lock".Sig, Q_DELAY =>, ACK_REQ => "Sfty_Status"."200RU01-QQ03_Lock".AckReq, DIAG =>)
   END_RUNG
   // the same network as SCL:
   #"SF_200RU01-QQ03_lock"(E_STOP := "I_200KF04BusModuleF"."1_LM.FI_UK",   // ESTOP1
                           ACK := "Sfty_InterfaceSfty"."200RU01-QQ03_In".Ack,
                           Q => "Sfty_Status"."200RU01-QQ03_Lock".Sig,
                           ACK_REQ => "Sfty_Status"."200RU01-QQ03_Lock".AckReq);
END_REGION

REGION Network 63: 200RU01-QQ04 - gate is closed and locked
   RUNG wire#powerrail
      #"SF_200RU01-QQ04_lock".ESTOP1(E_STOP := "I_200KF04BusModuleF"."3_LM.FI_UK", ACK_NEC :=, ACK := "Sfty_InterfaceSfty"."200RU01-QQ04_In".Ack, TIME_DEL :=, Q => "Sfty_Status"."200RU01-QQ04_Lock".Sig, Q_DELAY =>, ACK_REQ => "Sfty_Status"."200RU01-QQ04_Lock".AckReq, DIAG =>)
   END_RUNG
   // the same network as SCL:
   #"SF_200RU01-QQ04_lock"(E_STOP := "I_200KF04BusModuleF"."3_LM.FI_UK",   // ESTOP1
                           ACK := "Sfty_InterfaceSfty"."200RU01-QQ04_In".Ack,
                           Q => "Sfty_Status"."200RU01-QQ04_Lock".Sig,
                           ACK_REQ => "Sfty_Status"."200RU01-QQ04_Lock".AckReq);
END_REGION

REGION Network 64: 200RU01-QQ05 - gate is closed and locked
   RUNG wire#powerrail
      #"SF_200RU01-QQ05_lock".ESTOP1(E_STOP := "I_200KF03BusModuleF"."1_LM.FI_UK", ACK_NEC :=, ACK := "Sfty_InterfaceSfty"."200RU01-QQ05_In".Ack, TIME_DEL :=, Q => "Sfty_Status"."200RU01-QQ05_Lock".Sig, Q_DELAY =>, ACK_REQ => "Sfty_Status"."200RU01-QQ05_Lock".AckReq, DIAG =>)
   END_RUNG
   // the same network as SCL:
   #"SF_200RU01-QQ05_lock"(E_STOP := "I_200KF03BusModuleF"."1_LM.FI_UK",   // ESTOP1
                           ACK := "Sfty_InterfaceSfty"."200RU01-QQ05_In".Ack,
                           Q => "Sfty_Status"."200RU01-QQ05_Lock".Sig,
                           ACK_REQ => "Sfty_Status"."200RU01-QQ05_Lock".AckReq);
END_REGION

REGION Network 65: 100+RU01-BG01 - fence 1 is closed
   RUNG wire#powerrail
      #"SF_100+RU01-BG01_close".ESTOP1(E_STOP := "100RU01-BG01_4", ACK_NEC :=, ACK := "Sfty_InterfaceSfty".Ack.Group01, TIME_DEL :=, Q => "Sfty_Status"."100RU01-BG01_4_Fence".Sig, Q_DELAY =>, ACK_REQ => "Sfty_Status"."100RU01-BG01_4_Fence".AckReq, DIAG =>)
   END_RUNG
   // the same network as SCL:
   #"SF_100+RU01-BG01_close"(E_STOP := "100RU01-BG01_4",   // ESTOP1
                           ACK := "Sfty_InterfaceSfty".Ack.Group01,
                           Q => "Sfty_Status"."100RU01-BG01_4_Fence".Sig,
                           ACK_REQ => "Sfty_Status"."100RU01-BG01_4_Fence".AckReq);
END_REGION

REGION Network 66: 100+RU01-BG02 - fence 2 is closed
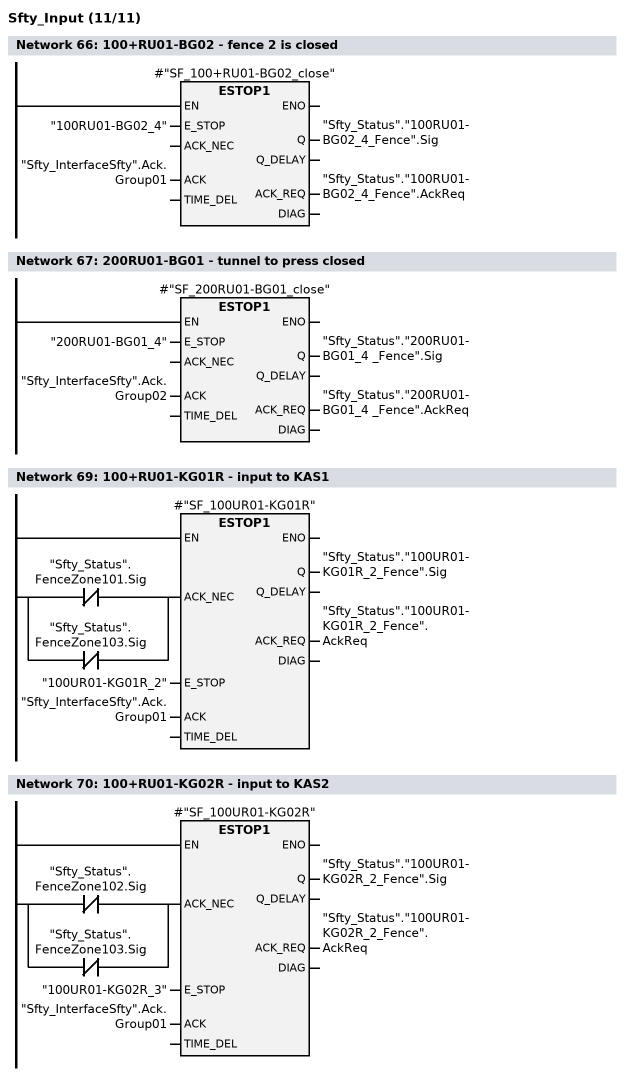
   RUNG wire#powerrail
      #"SF_100+RU01-BG02_close".ESTOP1(E_STOP := "100RU01-BG02_4", ACK_NEC :=, ACK := "Sfty_InterfaceSfty".Ack.Group01, TIME_DEL :=, Q => "Sfty_Status"."100RU01-BG02_4_Fence".Sig, Q_DELAY =>, ACK_REQ => "Sfty_Status"."100RU01-BG02_4_Fence".AckReq, DIAG =>)
   END_RUNG
   // the same network as SCL:
   #"SF_100+RU01-BG02_close"(E_STOP := "100RU01-BG02_4",   // ESTOP1
                           ACK := "Sfty_InterfaceSfty".Ack.Group01,
                           Q => "Sfty_Status"."100RU01-BG02_4_Fence".Sig,
                           ACK_REQ => "Sfty_Status"."100RU01-BG02_4_Fence".AckReq);
END_REGION

REGION Network 67: 200RU01-BG01 - tunnel to press closed
   RUNG wire#powerrail
      #"SF_200RU01-BG01_close".ESTOP1(E_STOP := "200RU01-BG01_4", ACK_NEC :=, ACK := "Sfty_InterfaceSfty".Ack.Group02, TIME_DEL :=, Q => "Sfty_Status"."200RU01-BG01_4 _Fence".Sig, Q_DELAY =>, ACK_REQ => "Sfty_Status"."200RU01-BG01_4 _Fence".AckReq, DIAG =>)
   END_RUNG
   // the same network as SCL:
   #"SF_200RU01-BG01_close"(E_STOP := "200RU01-BG01_4",   // ESTOP1
                           ACK := "Sfty_InterfaceSfty".Ack.Group02,
                           Q => "Sfty_Status"."200RU01-BG01_4 _Fence".Sig,
                           ACK_REQ => "Sfty_Status"."200RU01-BG01_4 _Fence".AckReq);
END_REGION

REGION Network 68: *************** Light barriers ***************
END_REGION

REGION Network 69: 100+RU01-KG01R - input to KAS1
   RUNG wire#powerrail
      #"SF_100UR01-KG01R".ESTOP1(ACK_NEC := wire#w1, E_STOP := "100UR01-KG01R_2", ACK := "Sfty_InterfaceSfty".Ack.Group01, TIME_DEL :=, Q => "Sfty_Status"."100UR01-KG01R_2_Fence".Sig, Q_DELAY =>, ACK_REQ => "Sfty_Status"."100UR01-KG01R_2_Fence".AckReq, DIAG =>)
   END_RUNG
   RUNG wire#powerrail
      I_Contact( "Sfty_Status".FenceZone101.Sig )
   END_RUNG wire#w1
   RUNG wire#powerrail
      I_Contact( "Sfty_Status".FenceZone103.Sig )
   END_RUNG wire#w1
   // the same network as SCL:
   #"SF_100UR01-KG01R"(ACK_NEC := NOT "Sfty_Status".FenceZone101.Sig OR NOT "Sfty_Status".FenceZone103.Sig,   // ESTOP1
                       E_STOP := "100UR01-KG01R_2",
                       ACK := "Sfty_InterfaceSfty".Ack.Group01,
                       Q => "Sfty_Status"."100UR01-KG01R_2_Fence".Sig,
                       ACK_REQ => "Sfty_Status"."100UR01-KG01R_2_Fence".AckReq);
END_REGION

REGION Network 70: 100+RU01-KG02R - input to KAS2
   RUNG wire#powerrail
      #"SF_100UR01-KG02R".ESTOP1(ACK_NEC := wire#w1, E_STOP := "100UR01-KG02R_3", ACK := "Sfty_InterfaceSfty".Ack.Group01, TIME_DEL :=, Q => "Sfty_Status"."100UR01-KG02R_2_Fence".Sig, Q_DELAY =>, ACK_REQ => "Sfty_Status"."100UR01-KG02R_2_Fence".AckReq, DIAG =>)
   END_RUNG
   RUNG wire#powerrail
      I_Contact( "Sfty_Status".FenceZone102.Sig )
   END_RUNG wire#w1
   RUNG wire#powerrail
      I_Contact( "Sfty_Status".FenceZone103.Sig )
   END_RUNG wire#w1
   // the same network as SCL:
   #"SF_100UR01-KG02R"(ACK_NEC := NOT "Sfty_Status".FenceZone102.Sig OR NOT "Sfty_Status".FenceZone103.Sig,   // ESTOP1
                       E_STOP := "100UR01-KG02R_3",
                       ACK := "Sfty_InterfaceSfty".Ack.Group01,
                       Q => "Sfty_Status"."100UR01-KG02R_2_Fence".Sig,
                       ACK_REQ => "Sfty_Status"."100UR01-KG02R_2_Fence".AckReq);
END_REGION

REGION Network 71: *************** EDM function ***************
END_REGION

REGION Network 72: *************** Reserves ***************
END_REGION
END_FUNCTION_BLOCK
